// TIA Portal V17 export
// export: Created 2022-04-06T07:28:39.3100939Z, ExportSetting WithDefaults, DisplayName Totally Integrated Automation Portal, DisplayVersion V17, DisplayName TIA Portal Openness, DisplayVersion V17, DisplayName TIA Portal Version Control Interface, DisplayVersion V17, DisplayName TIA Portal Test Suite Advanced, DisplayVersion V17, DisplayName SINAMICS Startdrive Advanced, DisplayVersion V17, DisplayName SINAMICS Startdrive G130, G150, S120, S150, SINAMICS MV, S210, DisplayVersion V17, DisplayName SINAMICS Startdrive G110M, G120, G120C, G120D, G120P, G115D, DisplayVersion V17, DisplayName STEP 7 Professional, DisplayVersion V17, DisplayName STEP 7 Safety, DisplayVersion V17, DisplayName WinCC Advanced / Unified PC, DisplayVersion V17
DATA_BLOCK "Data"   // DB147
{ S7_Optimized_Access := 'TRUE' }
VERSION : 0.1
// stored: AutoNumber true, DBAccessibleFromOPCUA true, DBAccessibleFromWebserver true, IsOnlyStoredInLoadMemory false, IsRetainMemResEnabled false, IsWriteProtectedInAS false, MemoryReserve 100
   VAR
      rdSysT { ExternalWritable := 'False'} : Struct
         retVal { ExternalWritable := 'False'} : Int;   // return value
         "time" { ExternalWritable := 'False'} : DTL;   // system time
      END_STRUCT;
      simulation : Struct
         amplitude : Real := 6.0;   // Amplitude
         offset : Real := -22.0;   // Offset
         periode : UDInt := 60000;   // Periode in milliseconds
         value { ExternalWritable := 'False'} : Real;   // Calculated Sinus value / Calculated Sinus values
      END_STRUCT;
   END_VAR
   VAR RETAIN
      write : Bool;   // trigger for data logging
      dataLogSameFile : Struct
         enable : Bool := TRUE;   // TRUE: enable function block
         delete : Bool;   // TRUE: Delete data log(s)
         data : Struct   // data logging data
            temperature : Real;   // temperature to log
            Pressure : Real;
            Flow : Real;
         END_STRUCT;
         done { ExternalWritable := 'False'} : Bool;   // TRUE: Commanded functionality has been completed successfully
         error { ExternalWritable := 'False'} : Bool;   // TRUE: An error occurred during the execution of the FB
         status { ExternalWritable := 'False'} : Word;   // Status of the FB "DataLog1x00"
         subFunctionStatus { ExternalWritable := 'False'} : Word;   // Subfunction status
         numberRecords { ExternalWritable := 'False'} : UDInt;   // Current number of data records in the data log
         sync { ExternalWritable := 'False'} : Bool;   // "numberRecords" is synchronized
         last { ExternalWritable := 'False'} : Struct
            done { ExternalWritable := 'False'} : Struct
               old { ExternalAccessible := 'False'; ExternalVisible := 'False'; ExternalWritable := 'False'} : Bool;   // Old value for edge detection
               "time" { ExternalWritable := 'False'} : DTL;   // last time of successful completion
            END_STRUCT;
            error { ExternalWritable := 'False'} : Struct
               old { ExternalAccessible := 'False'; ExternalVisible := 'False'; ExternalWritable := 'False'} : Bool;   // Old value for edge detection
               "time" { ExternalWritable := 'False'} : DTL;   // last time of completion with error
               status { ExternalWritable := 'False'} : Word;   // 16#8601: DataLogCreate, 16#8602: DataLogOpen, 16#8603: DataLogWrite, 16#8604: DataLogClear, 16#8605: DataLogClose, 16#8606: DataLogNewFile, 16#8607: DataLogDelete
               subFunctionStatus { ExternalWritable := 'False'} : Word;   // Subfunction status
            END_STRUCT;
         END_STRUCT;
      END_STRUCT;
      tmailcAlarm : Struct
         enable : Bool := TRUE;   // TRUE: enable function block
         toS : String[240] := 'receiver@siemens.de';   // Recipient address
         mailAddrParam : TMail_QDN_SEC;   // addressing parameters
         done { ExternalWritable := 'False'} : Bool;   // E-mail has been sent
         error { ExternalWritable := 'False'} : Bool;   // Error while sending the e-mail
         status { ExternalWritable := 'False'} : Word;   // Status when error occured
         last { ExternalWritable := 'False'} : Struct
            done { ExternalWritable := 'False'} : Struct
               old { ExternalAccessible := 'False'; ExternalVisible := 'False'; ExternalWritable := 'False'} : Bool;   // Old value for edge detection
               "time" { ExternalWritable := 'False'} : DTL;   // last time of successful completion
            END_STRUCT;
            error { ExternalWritable := 'False'} : Struct
               old { ExternalAccessible := 'False'; ExternalVisible := 'False'; ExternalWritable := 'False'} : Bool;   // Old value for edge detection
               "time" { ExternalWritable := 'False'} : DTL;   // last time of completion with error
               status { ExternalWritable := 'False'} : Word;   // Status when error occured
               sfbStatus { ExternalWritable := 'False'} : Word;   // Error related SFB status
            END_STRUCT;
         END_STRUCT;
      END_STRUCT;
      dataLogNewFile : Struct
         enable : Bool := TRUE;   // TRUE: enable function block
         delete : Bool;   // TRUE: Delete data log(s)
         data : Struct   // data logging data
            temperature : Real;   // temperature to log
            Pressure : Real;
            Flow : Real;
         END_STRUCT;
         done { ExternalWritable := 'False'} : Bool;   // TRUE: Commanded functionality has been completed successfully
         error { ExternalWritable := 'False'} : Bool;   // TRUE: An error occurred during the execution of the FB
         status { ExternalWritable := 'False'} : Word;   // Status of the FB "DataLog1x00"
         subFunctionStatus { ExternalWritable := 'False'} : Word;   // Subfunction status
         id { ExternalWritable := 'False'} : DWord;   // Object ID of the data log
         numberRecords { ExternalWritable := 'False'} : UDInt;   // Current number of data records in the data log
         sync { ExternalWritable := 'False'} : Bool;   // "numberRecords" is synchronized
         full { ExternalWritable := 'False'} : Bool;   // The maximum number of data records is reached
         fullOld { ExternalWritable := 'False'} : Bool;   // Old value for edge detection
         currentName { ExternalWritable := 'False'} : String;   // Current data log file name
         last { ExternalWritable := 'False'} : Struct
            done { ExternalWritable := 'False'} : Struct
               old { ExternalAccessible := 'False'; ExternalVisible := 'False'; ExternalWritable := 'False'} : Bool;   // Old value for edge detection
               "time" { ExternalWritable := 'False'} : DTL;   // last time of successful completion
            END_STRUCT;
            error { ExternalWritable := 'False'} : Struct
               old { ExternalAccessible := 'False'; ExternalVisible := 'False'; ExternalWritable := 'False'} : Bool;   // Old value for edge detection
               "time" { ExternalWritable := 'False'} : DTL;   // last time of completion with error
               status { ExternalWritable := 'False'} : Word;   // 16#8601: DataLogCreate, 16#8602: DataLogOpen, 16#8603: DataLogWrite, 16#8604: DataLogClear, 16#8605: DataLogClose, 16#8606: DataLogNewFile, 16#8607: DataLogDelete
               subFunctionStatus { ExternalWritable := 'False'} : Word;   // Subfunction status
            END_STRUCT;
         END_STRUCT;
      END_STRUCT;
      tmailcCsvTransfer : Struct
         enable : Bool := TRUE;   // TRUE: enable function block
         toS : String[240] := 'receiver@siemens.de';   // Recipient address
         mailAddrParam : TMail_QDN_SEC;   // addressing parameters
         attachment : TMail_FileReference;   // Attachment
         done { ExternalWritable := 'False'} : Bool;   // E-mail has been sent
         error { ExternalWritable := 'False'} : Bool;   // Error while sending the e-mail
         status { ExternalWritable := 'False'} : Word;   // Status when error occured
         last { ExternalWritable := 'False'} : Struct
            done { ExternalWritable := 'False'} : Struct
               old { ExternalAccessible := 'False'; ExternalVisible := 'False'; ExternalWritable := 'False'} : Bool;   // Old value for edge detection
               "time" { ExternalWritable := 'False'} : DTL;   // last time of successful completion
            END_STRUCT;
            error { ExternalWritable := 'False'} : Struct
               old { ExternalAccessible := 'False'; ExternalVisible := 'False'; ExternalWritable := 'False'} : Bool;   // Old value for edge detection
               "time" { ExternalWritable := 'False'} : DTL;   // last time of completion with error
               status { ExternalWritable := 'False'} : Word;   // Status when error occured
               sfbStatus { ExternalWritable := 'False'} : Word;   // Error related SFB status
            END_STRUCT;
         END_STRUCT;
      END_STRUCT;
   END_VAR
BEGIN
   tmailcAlarm.mailAddrParam.InterfaceId := 64;
   tmailcAlarm.mailAddrParam.ID := 1;
   tmailcAlarm.mailAddrParam.ConnectionType := 16#22;
   tmailcAlarm.mailAddrParam.WatchDogTime := T#60s;
   tmailcAlarm.mailAddrParam.MailServerQDN := 'smtp.gmail.com.';
   tmailcAlarm.mailAddrParam.UserName := 'sender@googlemail.com';
   tmailcAlarm.mailAddrParam.PassWord := 'Password';
   tmailcAlarm.mailAddrParam.From.LocalPartPlusAtSign := 'sender@';
   tmailcAlarm.mailAddrParam.From.FullQualifiedDomainName := 'googlemail.com';
   tmailcAlarm.mailAddrParam.RemotePort := 587;
   tmailcAlarm.mailAddrParam.ActivateSecureConn := true;
   tmailcAlarm.mailAddrParam.TLSServerCertRef := 43;
   tmailcCsvTransfer.mailAddrParam.InterfaceId := 64;
   tmailcCsvTransfer.mailAddrParam.ID := 2;
   tmailcCsvTransfer.mailAddrParam.ConnectionType := 16#22;
   tmailcCsvTransfer.mailAddrParam.WatchDogTime := T#60s;
   tmailcCsvTransfer.mailAddrParam.MailServerQDN := 'smtp.gmail.com.';
   tmailcCsvTransfer.mailAddrParam.UserName := 'sender@googlemail.com';
   tmailcCsvTransfer.mailAddrParam.PassWord := 'Password';
   tmailcCsvTransfer.mailAddrParam.From.LocalPartPlusAtSign := 'sender@';
   tmailcCsvTransfer.mailAddrParam.From.FullQualifiedDomainName := 'googlemail.com';
   tmailcCsvTransfer.mailAddrParam.RemotePort := 587;
   tmailcCsvTransfer.mailAddrParam.ActivateSecureConn := true;
   tmailcCsvTransfer.mailAddrParam.TLSServerCertRef := 43;
   tmailcCsvTransfer.attachment.DirectoryPath := '/DataLogs/';
   tmailcCsvTransfer.attachment.FileName := 'datalog.csv';
END_DATA_BLOCK
